// TIA Portal V17 export
// export: Created 2025-04-09T08:02:53.9893687Z, ExportSetting WithDefaults, DisplayName Totally Integrated Automation Portal, DisplayVersion V17 Update 8, DisplayName TIA Portal Openness, DisplayVersion V17 Update 8, DisplayName TIA Portal Version Control Interface, DisplayVersion V17, DisplayName SINAMICS Startdrive Advanced, DisplayVersion V17 SP2, DisplayName SINAMICS Startdrive G110M, G120, G120C, G120D, G120P, G115D, DisplayVersion V17 SP2, DisplayName SINAMICS Startdrive G130, G150, S120, S150, SINAMICS MV, S210, DisplayVersion V17 SP2, DisplayName STEP 7 Professional, DisplayVersion V17 Update 8, DisplayName SINUMERIK ONE STEP 7 Toolbox, DisplayVersion V17 Update 12, DisplayName SINUMERIK ONE PLC Basic Program Plus, DisplayVersion V17 Update 12, DisplayName SINUMERIK 840D sl STEP 7 Toolbox, DisplayVersion V17 Update 12, DisplayName STEP 7 Safety, DisplayVersion V17 Update 6, DisplayName WinCC Advanced, DisplayVersion V17 Update 8
FUNCTION "FC7321_ROBOT_CELL_LOAD_FIXTURE" : Void   // FC7321, LAD
{ S7_Optimized_Access := 'FALSE' }
AUTHOR : ETXETAR
VERSION : 1.0
// stored: AutoNumber false, IsIECCheckEnabled false, SetENOAutomatically false, UDAEnableTagReadback false
   VAR_TEMP
      STATUS_BLKMOV : Int;
      TEMPORARY_I : Any;
      ZERO : Byte;   // ZERO
      STATUS_FILL : Int;   // STATUS FILL
   END_VAR
   VAR_TEMP   // added for the SCL form of the ladder/FBD networks
      _w1 : Bool;
   END_VAR
BEGIN

REGION Network 1: >>>>>>>>>>>>>> UNIT 01 <<<<<<<<<<<<<<
END_REGION

REGION Network 2: PART A LOADED
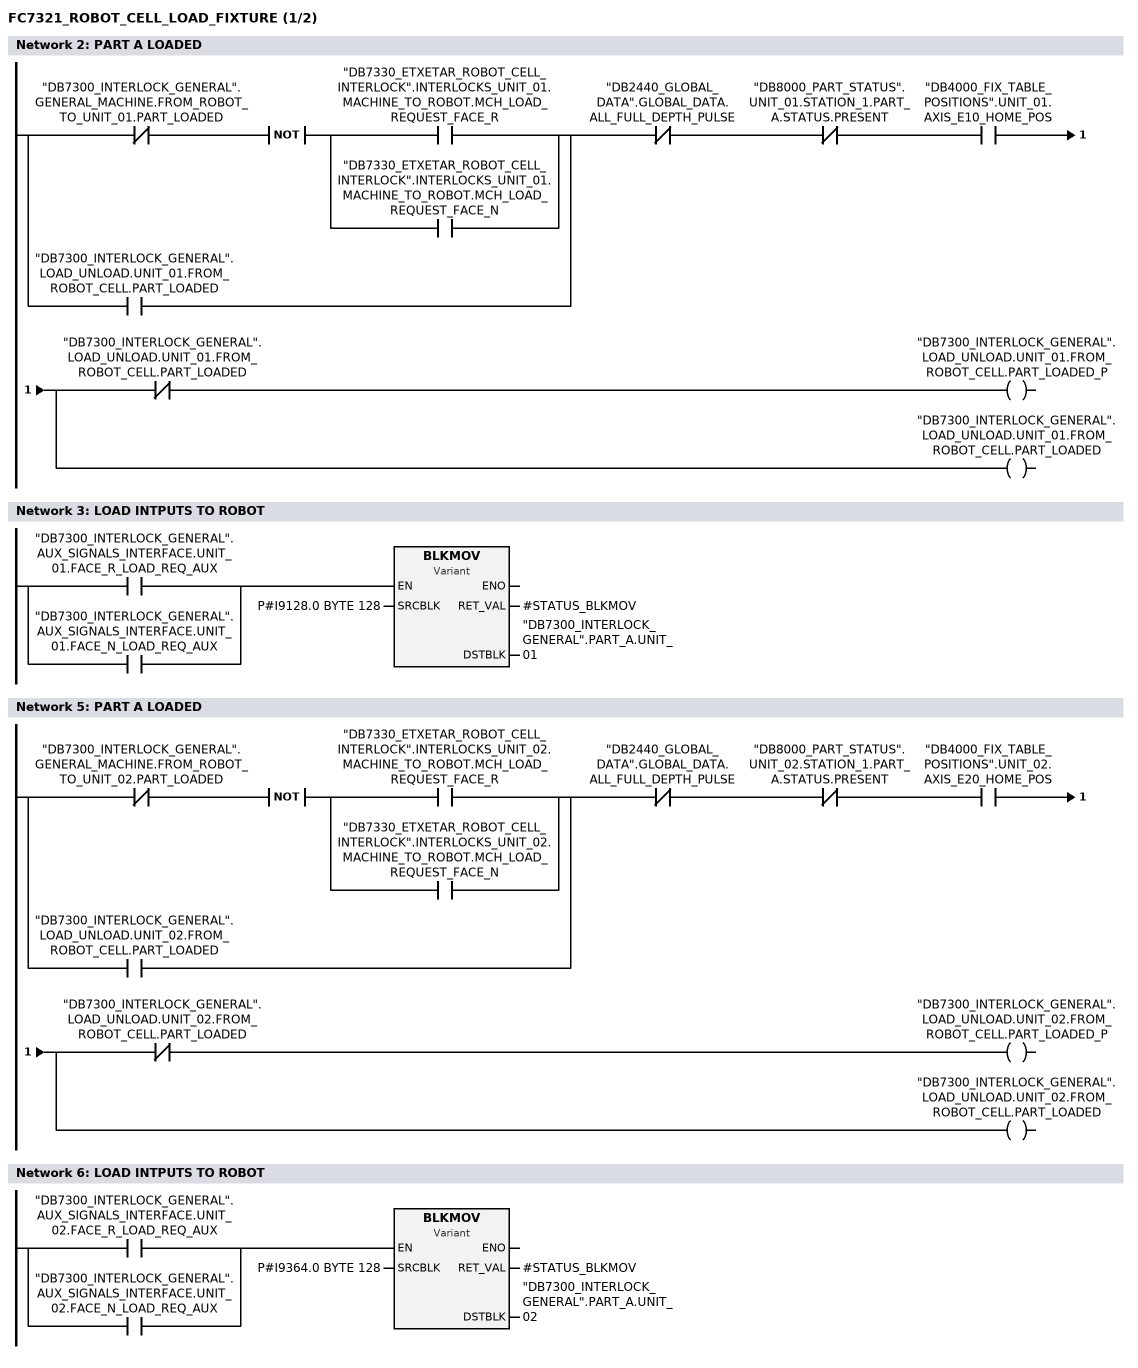
   RUNG wire#powerrail
      I_Contact( "DB7300_INTERLOCK_GENERAL".GENERAL_MACHINE.FROM_ROBOT_TO_UNIT_01.PART_LOADED )
      Not()
      wire#w1
      Contact( "DB7330_ETXETAR_ROBOT_CELL_INTERLOCK".INTERLOCKS_UNIT_01.MACHINE_TO_ROBOT.MCH_LOAD_REQUEST_FACE_R )
      wire#w2
      I_Contact( "DB2440_GLOBAL_DATA".GLOBAL_DATA.ALL_FULL_DEPTH_PULSE )
      I_Contact( "DB8000_PART_STATUS".UNIT_01.STATION_1.PART_A.STATUS.PRESENT )
      Contact( "DB4000_FIX_TABLE_POSITIONS".UNIT_01.AXIS_E10_HOME_POS )
      wire#w3
      I_Contact( "DB7300_INTERLOCK_GENERAL".LOAD_UNLOAD.UNIT_01.FROM_ROBOT_CELL.PART_LOADED )
      Coil( "DB7300_INTERLOCK_GENERAL".LOAD_UNLOAD.UNIT_01.FROM_ROBOT_CELL.PART_LOADED_P )
   END_RUNG
   RUNG wire#w1
      Contact( "DB7330_ETXETAR_ROBOT_CELL_INTERLOCK".INTERLOCKS_UNIT_01.MACHINE_TO_ROBOT.MCH_LOAD_REQUEST_FACE_N )
   END_RUNG wire#w2
   RUNG wire#powerrail
      Contact( "DB7300_INTERLOCK_GENERAL".LOAD_UNLOAD.UNIT_01.FROM_ROBOT_CELL.PART_LOADED )
   END_RUNG wire#w2
   RUNG wire#w3
      Coil( "DB7300_INTERLOCK_GENERAL".LOAD_UNLOAD.UNIT_01.FROM_ROBOT_CELL.PART_LOADED )
   END_RUNG
   // the same network as SCL:
   #_w1 := ((NOT (NOT "DB7300_INTERLOCK_GENERAL".GENERAL_MACHINE.FROM_ROBOT_TO_UNIT_01.PART_LOADED) AND ("DB7330_ETXETAR_ROBOT_CELL_INTERLOCK".INTERLOCKS_UNIT_01.MACHINE_TO_ROBOT.MCH_LOAD_REQUEST_FACE_R OR "DB7330_ETXETAR_ROBOT_CELL_INTERLOCK".INTERLOCKS_UNIT_01.MACHINE_TO_ROBOT.MCH_LOAD_REQUEST_FACE_N)) OR "DB7300_INTERLOCK_GENERAL".LOAD_UNLOAD.UNIT_01.FROM_ROBOT_CELL.PART_LOADED) AND NOT "DB2440_GLOBAL_DATA".GLOBAL_DATA.ALL_FULL_DEPTH_PULSE AND NOT "DB8000_PART_STATUS".UNIT_01.STATION_1.PART_A.STATUS.PRESENT AND "DB4000_FIX_TABLE_POSITIONS".UNIT_01.AXIS_E10_HOME_POS;
   "DB7300_INTERLOCK_GENERAL".LOAD_UNLOAD.UNIT_01.FROM_ROBOT_CELL.PART_LOADED_P := #_w1 AND NOT "DB7300_INTERLOCK_GENERAL".LOAD_UNLOAD.UNIT_01.FROM_ROBOT_CELL.PART_LOADED;
   "DB7300_INTERLOCK_GENERAL".LOAD_UNLOAD.UNIT_01.FROM_ROBOT_CELL.PART_LOADED := #_w1;
END_REGION

REGION Network 3: LOAD INTPUTS TO ROBOT
   RUNG wire#powerrail
      Contact( "DB7300_INTERLOCK_GENERAL".AUX_SIGNALS_INTERFACE.UNIT_01.FACE_R_LOAD_REQ_AUX )
      wire#w1
      { S7_Templates := "blk_type := Variant" } BLKMOV(SRCBLK := P#I9128.0 BYTE 128, RET_VAL => #STATUS_BLKMOV, DSTBLK => "DB7300_INTERLOCK_GENERAL".PART_A.UNIT_01)
   END_RUNG
   RUNG wire#powerrail
      Contact( "DB7300_INTERLOCK_GENERAL".AUX_SIGNALS_INTERFACE.UNIT_01.FACE_N_LOAD_REQ_AUX )
   END_RUNG wire#w1
   // the same network as SCL:
   IF "DB7300_INTERLOCK_GENERAL".AUX_SIGNALS_INTERFACE.UNIT_01.FACE_R_LOAD_REQ_AUX OR "DB7300_INTERLOCK_GENERAL".AUX_SIGNALS_INTERFACE.UNIT_01.FACE_N_LOAD_REQ_AUX THEN
       #STATUS_BLKMOV := BLKMOV(SRCBLK := P#I9128.0 BYTE 128, DSTBLK => "DB7300_INTERLOCK_GENERAL".PART_A.UNIT_01);
   END_IF;
END_REGION

REGION Network 4: >>>>>>>>>>>>>> UNIT 02 <<<<<<<<<<<<<<
END_REGION

REGION Network 5: PART A LOADED
   RUNG wire#powerrail
      I_Contact( "DB7300_INTERLOCK_GENERAL".GENERAL_MACHINE.FROM_ROBOT_TO_UNIT_02.PART_LOADED )
      Not()
      wire#w1
      Contact( "DB7330_ETXETAR_ROBOT_CELL_INTERLOCK".INTERLOCKS_UNIT_02.MACHINE_TO_ROBOT.MCH_LOAD_REQUEST_FACE_R )
      wire#w2
      I_Contact( "DB2440_GLOBAL_DATA".GLOBAL_DATA.ALL_FULL_DEPTH_PULSE )
      I_Contact( "DB8000_PART_STATUS".UNIT_02.STATION_1.PART_A.STATUS.PRESENT )
      Contact( "DB4000_FIX_TABLE_POSITIONS".UNIT_02.AXIS_E20_HOME_POS )
      wire#w3
      I_Contact( "DB7300_INTERLOCK_GENERAL".LOAD_UNLOAD.UNIT_02.FROM_ROBOT_CELL.PART_LOADED )
      Coil( "DB7300_INTERLOCK_GENERAL".LOAD_UNLOAD.UNIT_02.FROM_ROBOT_CELL.PART_LOADED_P )
   END_RUNG
   RUNG wire#w1
      Contact( "DB7330_ETXETAR_ROBOT_CELL_INTERLOCK".INTERLOCKS_UNIT_02.MACHINE_TO_ROBOT.MCH_LOAD_REQUEST_FACE_N )
   END_RUNG wire#w2
   RUNG wire#powerrail
      Contact( "DB7300_INTERLOCK_GENERAL".LOAD_UNLOAD.UNIT_02.FROM_ROBOT_CELL.PART_LOADED )
   END_RUNG wire#w2
   RUNG wire#w3
      Coil( "DB7300_INTERLOCK_GENERAL".LOAD_UNLOAD.UNIT_02.FROM_ROBOT_CELL.PART_LOADED )
   END_RUNG
   // the same network as SCL:
   #_w1 := ((NOT (NOT "DB7300_INTERLOCK_GENERAL".GENERAL_MACHINE.FROM_ROBOT_TO_UNIT_02.PART_LOADED) AND ("DB7330_ETXETAR_ROBOT_CELL_INTERLOCK".INTERLOCKS_UNIT_02.MACHINE_TO_ROBOT.MCH_LOAD_REQUEST_FACE_R OR "DB7330_ETXETAR_ROBOT_CELL_INTERLOCK".INTERLOCKS_UNIT_02.MACHINE_TO_ROBOT.MCH_LOAD_REQUEST_FACE_N)) OR "DB7300_INTERLOCK_GENERAL".LOAD_UNLOAD.UNIT_02.FROM_ROBOT_CELL.PART_LOADED) AND NOT "DB2440_GLOBAL_DATA".GLOBAL_DATA.ALL_FULL_DEPTH_PULSE AND NOT "DB8000_PART_STATUS".UNIT_02.STATION_1.PART_A.STATUS.PRESENT AND "DB4000_FIX_TABLE_POSITIONS".UNIT_02.AXIS_E20_HOME_POS;
   "DB7300_INTERLOCK_GENERAL".LOAD_UNLOAD.UNIT_02.FROM_ROBOT_CELL.PART_LOADED_P := #_w1 AND NOT "DB7300_INTERLOCK_GENERAL".LOAD_UNLOAD.UNIT_02.FROM_ROBOT_CELL.PART_LOADED;
   "DB7300_INTERLOCK_GENERAL".LOAD_UNLOAD.UNIT_02.FROM_ROBOT_CELL.PART_LOADED := #_w1;
END_REGION

REGION Network 6: LOAD INTPUTS TO ROBOT
   RUNG wire#powerrail
      Contact( "DB7300_INTERLOCK_GENERAL".AUX_SIGNALS_INTERFACE.UNIT_02.FACE_R_LOAD_REQ_AUX )
      wire#w1
      { S7_Templates := "blk_type := Variant" } BLKMOV(SRCBLK := P#I9364.0 BYTE 128, RET_VAL => #STATUS_BLKMOV, DSTBLK => "DB7300_INTERLOCK_GENERAL".PART_A.UNIT_02)
   END_RUNG
   RUNG wire#powerrail
      Contact( "DB7300_INTERLOCK_GENERAL".AUX_SIGNALS_INTERFACE.UNIT_02.FACE_N_LOAD_REQ_AUX )
   END_RUNG wire#w1
   // the same network as SCL:
   IF "DB7300_INTERLOCK_GENERAL".AUX_SIGNALS_INTERFACE.UNIT_02.FACE_R_LOAD_REQ_AUX OR "DB7300_INTERLOCK_GENERAL".AUX_SIGNALS_INTERFACE.UNIT_02.FACE_N_LOAD_REQ_AUX THEN
       #STATUS_BLKMOV := BLKMOV(SRCBLK := P#I9364.0 BYTE 128, DSTBLK => "DB7300_INTERLOCK_GENERAL".PART_A.UNIT_02);
   END_IF;
END_REGION

REGION Network 7: >>>>>>>>>>>>>> UNIT 03 MEASURING STATION <<<<<<<<<<<<<<
END_REGION

REGION Network 8: PART A LOADED
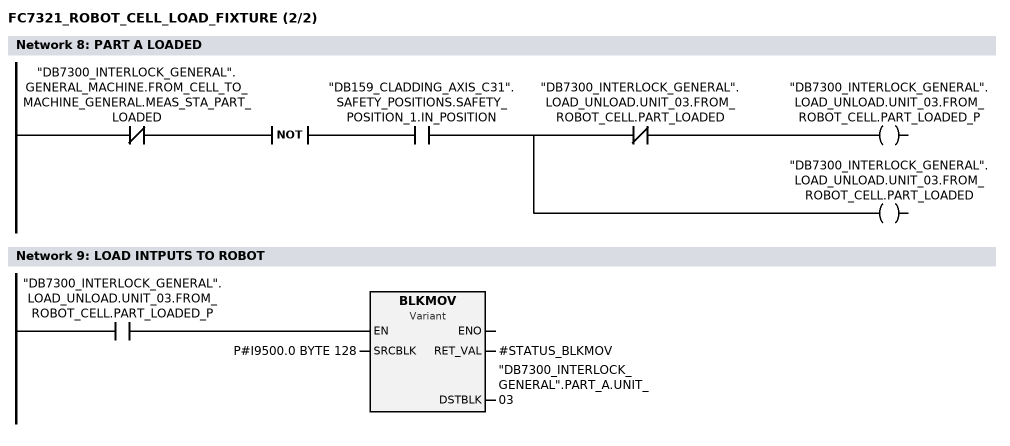
   RUNG wire#powerrail
      I_Contact( "DB7300_INTERLOCK_GENERAL".GENERAL_MACHINE.FROM_CELL_TO_MACHINE_GENERAL.MEAS_STA_PART_LOADED )
      Not()
      Contact( "DB159_CLADDING_AXIS_C31".SAFETY_POSITIONS.SAFETY_POSITION_1.IN_POSITION )
      wire#w1
      I_Contact( "DB7300_INTERLOCK_GENERAL".LOAD_UNLOAD.UNIT_03.FROM_ROBOT_CELL.PART_LOADED )
      Coil( "DB7300_INTERLOCK_GENERAL".LOAD_UNLOAD.UNIT_03.FROM_ROBOT_CELL.PART_LOADED_P )
   END_RUNG
   RUNG wire#w1
      Coil( "DB7300_INTERLOCK_GENERAL".LOAD_UNLOAD.UNIT_03.FROM_ROBOT_CELL.PART_LOADED )
   END_RUNG
   // the same network as SCL:
   #_w1 := NOT (NOT "DB7300_INTERLOCK_GENERAL".GENERAL_MACHINE.FROM_CELL_TO_MACHINE_GENERAL.MEAS_STA_PART_LOADED) AND "DB159_CLADDING_AXIS_C31".SAFETY_POSITIONS.SAFETY_POSITION_1.IN_POSITION;
   "DB7300_INTERLOCK_GENERAL".LOAD_UNLOAD.UNIT_03.FROM_ROBOT_CELL.PART_LOADED_P := #_w1 AND NOT "DB7300_INTERLOCK_GENERAL".LOAD_UNLOAD.UNIT_03.FROM_ROBOT_CELL.PART_LOADED;
   "DB7300_INTERLOCK_GENERAL".LOAD_UNLOAD.UNIT_03.FROM_ROBOT_CELL.PART_LOADED := #_w1;
END_REGION

REGION Network 9: LOAD INTPUTS TO ROBOT
   RUNG wire#powerrail
      Contact( "DB7300_INTERLOCK_GENERAL".LOAD_UNLOAD.UNIT_03.FROM_ROBOT_CELL.PART_LOADED_P )
      { S7_Templates := "blk_type := Variant" } BLKMOV(SRCBLK := P#I9500.0 BYTE 128, RET_VAL => #STATUS_BLKMOV, DSTBLK => "DB7300_INTERLOCK_GENERAL".PART_A.UNIT_03)
   END_RUNG
   // the same network as SCL:
   IF "DB7300_INTERLOCK_GENERAL".LOAD_UNLOAD.UNIT_03.FROM_ROBOT_CELL.PART_LOADED_P THEN
       #STATUS_BLKMOV := BLKMOV(SRCBLK := P#I9500.0 BYTE 128, DSTBLK => "DB7300_INTERLOCK_GENERAL".PART_A.UNIT_03);
   END_IF;
END_REGION
END_FUNCTION
